(* IEC 61131-3 sources: test_training/GmpAccess2/src, 3 files *)

(* ---- EasyProg.st ---- *)
PROGRAM EasyProg
VAR
	i	: INT;
	str	: STRING(123);
END_VAR

i := i + 1;

str := 'Mein Text!';
i := renameFunction(in := i);

END_PROGRAM

(* ---- ScopeProg.st ---- *)
(* program to handle scope recordings *)
PROGRAM ScopeProg
VAR
	pLockHandle : UDINT;
	retVal 		: GMP232X_RETVAL;
END_VAR

updateScopeState();

IF triggerScope THEN
	triggerScopeIfPossible();
END_IF

IF exportScope THEN
	exportScopeIfReady();
END_IF

END_PROGRAM

ACTIONS

	(* reset scope trigger flag and trigger scope if possible *)
	ACTION triggerScopeIfPossible
		triggerScope := FALSE;
		IF scopeState.State = GMP232X_SCOPE_STATE_NOTTRIGGERED OR
				scopeState.State = GMP232X_SCOPE_STATE_READY THEN
			GMP232X_TRIGGERSCOPE(MODULE_NUMBER, 0);
		END_IF
	END_ACTION

	(* reset export scope flag and export scope to path if recording is ready *)
	ACTION exportScopeIfReady
		exportScope := FALSE;
		IF (UDINT_TO_DWORD(scopeState.State) AND GMP232X_SCOPE_STATE_NEWDATA) = GMP232X_SCOPE_STATE_NEWDATA THEN
			retVal := GMP232X_TAKESCOPELOCK(MODULE_NUMBER, 0, 3, ADR(pLockHandle));
			Util_LogWrn('Take Lock');
			Util_LogWrn(UDINT_TO_STRING(pLockHandle));
			logError(retVal);
			retVal := GMP232X_EXPORTSCOPE(MODULE_NUMBER, 0, pLockHandle, 'myScopeRecording', 0);
			logError(retVal);
			Util_LogWrn('Give Lock');
			Util_LogWrn(UDINT_TO_STRING(pLockHandle));
			retVal := GMP232X_GIVESCOPELOCK(MODULE_NUMBER, 0, pLockHandle);
			logError(retVal);
		END_IF
	END_ACTION

	(* update scope state *)
	ACTION updateScopeState
		GMP232X_GETSCOPESTATE(MODULE_NUMBER, 0, ADR(scopeState));
	END_ACTION

END_ACTIONS

(* ---- Values.st ---- *)
PROGRAM Values
VAR
	val : ARRAY [0..2] OF ChanValue;
	i : INT;
END_VAR

FOR i := 0 TO 2 DO
	val[i]();
END_FOR
;
END_PROGRAM

ACTIONS

END_ACTIONS
